SUBAPPLICATION Uebung_102b (* DigitalInput_I1 auf DigitalOutput_Q1/_Q2, mit Plug and Socket *)
  (* Standard: 61499-2; Description: Copyright (c) 2023 Meisterschulen am Ostbahnhof This program and the accompanying materials are made available under the terms of the Eclipse Public License 2.0 which is available at https://www.eclipse.org/legal/epl-2.0/ SPDX-License-Identifier: EPL-2.0 *)
  (* Version 1.0, 2023-10-23, Franz Höpfinger, Meisterschulen am Ostbahnhof *)
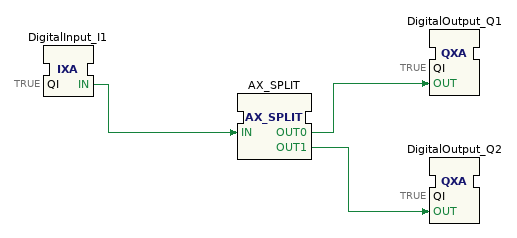
  FBS
    DigitalInput_I1 : IXA(QI := TRUE);
    DigitalOutput_Q1 : QXA(QI := TRUE);
    DigitalOutput_Q2 : QXA(QI := TRUE);
    AX_SPLIT : AX_SPLIT;
  END_FBS
  ADAPTER_CONNECTIONS
    DigitalInput_I1.IN TO AX_SPLIT.IN;
    AX_SPLIT.OUT0 TO DigitalOutput_Q1.OUT;
    AX_SPLIT.OUT1 TO DigitalOutput_Q2.OUT;
  END_CONNECTIONS
END_SUBAPPLICATION
